// What the runner knows about how long the current test has been going.
//
// Separate from the verdict surface because it has its own consumers: a teardown
// deciding how long to wait, a metrics sink, and AssertCompletedWithin - which is
// built on ElapsedCycles rather than on bookkeeping inside the test.
INTERFACE I_TestTiming EXTENDS __SYSTEM.IQueryInterface

// Scans consumed by this test so far, counted by the runner.
//
// The reproducible measure. Prefer it to ElapsedTime for anything asserted on.
PROPERTY ElapsedCycles : UDINT
GET
END_GET
END_PROPERTY

// Seconds elapsed. Wall clock, so it varies with jitter across Windows, BSD,
// Linux RT and containers - report it, but assert on ElapsedCycles.
// Seconds elapsed for this test. Pairs with ElapsedCycles - the same span
// measured two ways.
//
// Wall clock, so it varies with jitter across Windows, BSD, Linux RT and
// containers. Report it; assert on ElapsedCycles.
PROPERTY ElapsedTime : LREAL
GET
END_GET
END_PROPERTY

// TRUE on the first scan of the test body. The setup hook for anything not worth
// implementing I_TestSetup for.
PROPERTY IsFirstCycle : BOOL
GET
END_GET
END_PROPERTY

END_INTERFACE

(* stored: Version 1.1.0.1, ProductVersion 3.1.4026.18
   Itf I_TestTiming: Id {4c0ba300-c002-4276-b370-a1cbf88726a1}
   Property ElapsedCycles: Id {bc226552-2c19-4901-8c04-56eecc378b32}
   Get Get: Id {efdfccc1-5fb0-4bb7-8b31-559270d3eeb0}
   Property ElapsedTime: Id {a310d087-806e-40ae-90b2-2b65f6d71b3e}
   Get Get: Id {ab7541c9-a3ac-4056-9fc2-1926a021c61e}
   Property IsFirstCycle: Id {b49679d4-0653-4ed3-bc5f-2da428ccb0d3}
   Get Get: Id {167b4417-4b44-4915-8fac-c966dc3357c9} *)
